INTERFACE ILight

METHOD M_Off
END_METHOD

PROPERTY P_ControlValue : BOOL
SET
END_SET
GET
END_GET
END_PROPERTY

METHOD M_On
END_METHOD

METHOD M_Execution
END_METHOD

END_INTERFACE

(* stored: Version 1.1.0.1, ProductVersion 3.1.0.23
   Itf ILight: Id {3565a55e-14ef-499b-9ae1-18d8e4acc4c8}
   Method M_Off: Id {3803cdc9-dd34-4531-9d06-6c96402f42c7}
   Property P_ControlValue: Id {6e1157b2-5bf6-483c-a2fe-25c64b4ab075}
   Set Set: Id {7c7e8938-e5d1-4954-b4e5-17adf0402d3b}
   Get Get: Id {cfa9e474-1ee4-4804-ab55-2295e728314c}
   Method M_On: Id {cc65df01-5c0e-4d92-b648-2203af88d63c}
   Method M_Execution: Id {f2737487-df93-4ce7-bd45-f8f4c0002286} *)
